Staubli VAL3: IO.dtx

mdesc mNomSpeed
public dio diStart = {link=usrIn0}
public dio diStop
public dio diGanying
public dio diTab
public dio diXi
public dio dIn{}
  [dIn1] = {link=BasicIO-1\%I0}
  [dIn8] = {link=BasicIO-1\%I7}
  [dIn7] = {link=BasicIO-1\%I6}
  [dIn6] = {link=BasicIO-1\%I5}
  [dIn5] = {link=BasicIO-1\%I4}
  [dIn4] = {link=BasicIO-1\%I3}
  [dIn3] = {link=BasicIO-1\%I2}
  [dIn2] = {link=BasicIO-1\%I1}
  [dIn9] = {link=BasicIO-1\%I8}
  [dIn10] = {link=BasicIO-1\%I9}
  [dIn11] = {link=BasicIO-1\%I10}
  [dIn12] = {link=BasicIO-1\%I11}
  [dIn13] = {link=BasicIO-1\%I12}
  [dIn14] = {link=BasicIO-1\%I13}
  [dIn15] = {link=BasicIO-1\%I14}
  [dIn16] = {link=BasicIO-1\%I15}
public dio dOut{}
  [dOut1] = {link=BasicIO-1\%Q0}
  [dOut2] = {link=BasicIO-1\%Q1}
  [dOut3] = {link=BasicIO-1\%Q2}
  [dOut4] = {link=BasicIO-1\%Q3}
  [dOut5] = {link=BasicIO-1\%Q4}
  [dOut6] = {link=BasicIO-1\%Q5}
  [dOut7] = {link=BasicIO-1\%Q6}
  [dOut8] = {link=BasicIO-1\%Q7}
  [dOut9] = {link=BasicIO-1\%Q8}
  [dOut10] = {link=BasicIO-1\%Q9}
  [dOut11] = {link=BasicIO-1\%Q10}
  [dOut12] = {link=BasicIO-1\%Q11}
  [dOut13] = {link=BasicIO-1\%Q12}
  [dOut14] = {link=BasicIO-1\%Q13}
  [dOut15] = {link=BasicIO-1\%Q14}
  [dOut16] = {link=BasicIO-1\%Q15}
string sIOName
string sList
bool bListRefresh
bool bUserRefresh
bool bExit
num nType
num nSelected
string sItem
public dio diEndStop = {link=usrIn1}
